FUNCTION_BLOCK SS4_Raiser_n_Flipper (* Basic FB with empty ECC *)
  (* Standard: 61499-2 *)
  (* Version 1.0, 2025-08-24, DEVIASH *)
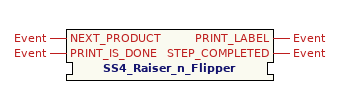
  EVENT_INPUT
    NEXT_PRODUCT;
    PRINT_IS_DONE;
  END_EVENT
  EVENT_OUTPUT
    PRINT_LABEL;
    STEP_COMPLETED;
  END_EVENT
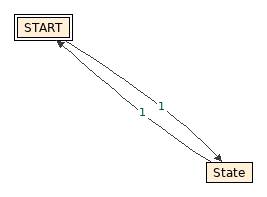
  EC_STATES
    START; (* Initial State *)
    State;
  END_STATES
  EC_TRANSITIONS
    START TO State := 1;
    State TO START := 1;
  END_TRANSITIONS
END_FUNCTION_BLOCK
